TYPE FB_ServoAchse_MoveAbs :
(
	UNDEFINIERT := 0,
	FB_MOVE_ABSOLUTE_1,
	FB_MOVE_ABSOLUTE_2
);
END_TYPE

(* stored: Version 1.1.0.1, ProductVersion 3.1.4018.5
   DUT FB_ServoAchse_MoveAbs: Id {cc00f0b3-836c-472b-aa67-4a3b2ebbd991} *)
